Universal Robots PolyScope program: L05_forcealign.urp

Program L05_forcealign (installation=default directory=/programs createdIn=5.9.1.1031110 lastSavedIn=5.9.1.1031110 robotSerialNumber=20195501059)
Calibrated DH parameters: a=[0.000146, -0.418764, -0.053981, 0.000058, -0.000023, 0]; d=[0.162545, 37.319448, -206.067439, 168.881546, 0.09955, 0.099464]; alpha=[1.57004, -0.001979, 0.002304, 1.570607, -1.57066, 0]; deltaTheta=[0, -0.174616, -1.258233, 1.432844, -0.000001, 0]
BeforeStart
  start_p := get_actual_tcp_pose()
  MoveL speed 250 mm/s, acceleration 1200 mm/s^2 (useActiveTCP=true) feature=Base
    Waypoint Waypoint (Variable): variable=start_p
Robot Program (runOnlyOnce=true)
  MoveL speed 250 mm/s, acceleration 1200 mm/s^2 (useActiveTCP=true) feature=Base
    Waypoint approach_p: TCP in base x=474.268 y=-600.261 z=130.712 mm, rx=-3.1089 ry=-0.0517 rz=-0.3637 rad; joints [113.688, -54.66, 72.57, -112.544, 282.504, 202.283] deg; TCP offset x=0 y=0 z=174 mm, rx=0 ry=0 rz=0 rad
    URCap Gripper (Robotiq_Grippers, Robotiq Inc.) dataModel(position=100.0, force=100.0, speed=100.0, positionInDouble=100.0, forceInDouble=100.0, speedInDouble=100.0, slaveIds=[9], blocking=true)
    MoveDirectionNode (selectedDirection=ZPlus toolParams=0.01, 0.6) feature=Joint_6_name
      Until TOOL_CONTACT_DETECTION (allowActions=false retraction=0 decelerationAcceleration=2 decelerationAngularAcceleration=34.906585)
    URCap Gripper (Robotiq_Grippers, Robotiq Inc.) dataModel(position=40.0, force=100.0, speed=100.0, positionInDouble=40.0, forceInDouble=100.0, speedInDouble=100.0, slaveIds=[9], blocking=true)
    MoveDirectionNode (selectedDirection=ZPlus toolParams=0.05, 0.6) feature=Joint_6_name
      Until DISTANCE (allowActions=false deceleration=3 distanceNodeType=STOP) Distance=0.035; motionParameters(blendRadius=0)
    URCap Zero FT Sensor (Robotiq_Copilot, Robotiq Inc.) dataModel(NodeInitializedKey=true, WaitForSteadyWrenchOptionKey=true)
    URCap Gripper (Robotiq_Grippers, Robotiq Inc.) dataModel(position=100.0, force=5.0, speed=30.0, positionInDouble=100.0, forceInDouble=5.0, speedInDouble=30.0, slaveIds=[9], blocking=true)
    Wait Sleep waitTime=2
    URCap Force Control (Robotiq_Copilot, Robotiq Inc.) dataModel(NodeInitializedKey=true, limit_x_neg=-100, limit_y_neg=-100, limit_z_neg=-100, limit_x_pos=100, limit_y_pos=100, limit_z_pos=100, limit_mx_neg=-20, limit_my_neg=-20, limit_mx_pos=20, limit_my_pos=20, stiffness_x=100, stiffness_y=100, stiffness_z_position=100, stiffness_mx=100, stiffness_my=100, stiffness_mz=100, limit_mz_neg=-90, limit_mz_pos=90, force_x=0, force_y=0, force_z=0, force_mx=0, force_my=0, force_mz=0, HackTriggeringContributionIsDefinedMethodKey=true, TranslatableFeatureKey=1, ft_control_x=true, adaptive_stiffness=true, ft_control_y=true, ft_control_z=true, ft_control_mx=true, ft_control_my=true, ft_control_mz=true, is_force_control_about_actual_position=true)
      Wait Sleep waitTime=3
    URCap Gripper (Robotiq_Grippers, Robotiq Inc.) dataModel(position=40.0, force=100.0, speed=100.0, positionInDouble=40.0, forceInDouble=100.0, speedInDouble=100.0, slaveIds=[9], blocking=true)
    MoveDirectionNode (selectedDirection=ZMinus) feature=Joint_6_name
      Until DISTANCE (allowActions=false deceleration=3 distanceNodeType=STOP) Distance=0.04; motionParameters(blendRadius=0)
